PROGRAM main
VAR
	GuardClosed AT %IX0.0 : bool;
	Start AT %IX0.1 : bool;
	MotorRun AT %QX0.0 : bool;
END_VAR

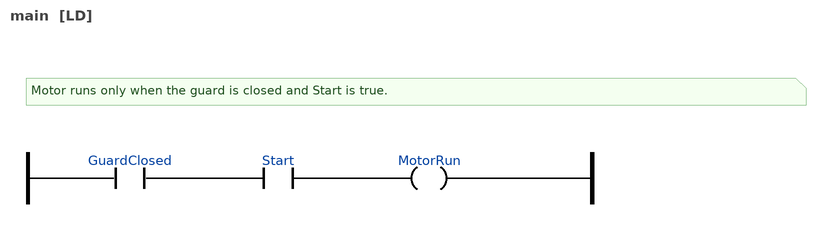
(* LD diagram, written out as Structured Text *)
(* Motor runs only when the guard is closed and Start is true. *)
MotorRun := GuardClosed AND Start;
END_PROGRAM
